/// Abstract base FB for components
{attribute 'enable_dynamic_creation' := ''}
{attribute 'reflection' := ''}
FUNCTION_BLOCK FB_ComponentBase IMPLEMENTS ITFComponent
VAR
	/// Unique ID of this instance (cam be used as index: P_ComponentPool.aComponents[iID]...)
	iId				: INT := -1;
	/// component active flag
	bActive			: BOOL;
	/// component state
	eState			: E_ComponentState;
	/// clear text info
	sClearText		: T_MaxString;
	/// last error debug info
	sLastError		: T_MaxString;	
	/// component type
	eTyp			: E_ComponentType;
	/// EventLog reference
	fbEventLog		: REFERENCE TO FB_EventLog;
	/// Last Event
	stLastEvent		: ST_Event;
	ptLastEvent		: POINTER TO ST_Event;
	
	
	/// Bereich
	eMachineArea	: E_MachineArea;
	/// component name
	sName			: STRING;
	/// BMK name
	sBMK			: STRING;
	/// path of this FB (e.g. for log: P_ComponentPool.fbVirtualMaster)
	{attribute 'no_init' := ''}
	{attribute 'instance-path' := ''}
	sPath			: STRING;	

END_VAR

///
/// Abstract base FB for components
/// TP/www.rmth.at/11.2014
///

/// Get's or set's a value indicating whether this component is active or not.
PROPERTY Active : BOOL
GET
Active := bActive;
END_GET
SET
bActive := Active;
sClearText := SEL(bActive, 'INACTIVE!', 'ACTIVE!');
END_SET
END_PROPERTY

PROPERTY BMK : STRING
GET
BMK := sBMK;
END_GET
SET
sBMK := BMK;
END_SET
END_PROPERTY

/// Get's value representing the component state.
PROPERTY ClearText : String
GET
ClearText := sClearText;
END_GET
END_PROPERTY

/// Unique component ID (cam be used as index: P_ComponentPool.aComponents[eID]...)
PROPERTY ID : INT
GET
ID := iId;
END_GET
SET
iID := Id;
END_SET
END_PROPERTY

/// Get's value representing the component state.
PROPERTY LastError : String
GET
LastError := sLastError;
END_GET
END_PROPERTY

PROPERTY MachineArea : E_MachineArea
GET
MachineArea := eMachineArea;
END_GET
SET
eMachineArea := MachineArea;
END_SET
END_PROPERTY

PROPERTY Name : STRING
GET
Name := sName;
END_GET
SET
sName := Name;
END_SET
END_PROPERTY

PROPERTY Path : String
GET
Path := sPath;
END_GET
END_PROPERTY

/// Reset component logic
{attribute 'object_name' := 'Reset'}
METHOD Reset
/// abstract base logic reset

sLastError := sEmpty;
MEMSET(ADR(stLastEvent), 0, SIZEOF(ST_EVENT));

// default: set state to ready
eState := E_ComponentState.eComponentState_ready;
END_METHOD

/// Run component logic
{attribute 'object_name' := 'Run'}
METHOD Run : E_ComponentState
/// abstract base logic run

// only rdy state may lead to run
IF eState = E_ComponentState.eComponentState_ready THEN
	eState := E_ComponentState.eComponentState_running;
END_IF

Run := eState;

IF stLastEvent.ePriority < E_Priority.ePriority_fault AND eState = E_ComponentState.eComponentState_error THEN
	WriteError(E_Event.eEvent_none, 'unbekannter Fehler');
END_IF
END_METHOD

/// Set EventLog reference
METHOD SetEventLogReference
VAR_IN_OUT
	/// HMI access provider.
	fbEventLogRef	: FB_EventLog;
END_VAR
fbEventLog REF= fbEventLogRef;
END_METHOD

/// Get's value representing the component state.
PROPERTY State : E_ComponentState
GET
State := eState;
END_GET
END_PROPERTY

/// Get's value representing the component state.
PROPERTY StateAsString : STRING
GET
CASE eState OF

	eComponentState_none :
		StateAsString := 'undefiniert';
	/// Component is resetting
	eComponentState_resetting:
		StateAsString := 'wird zurückgesetzt';
	/// Component is ready
	eComponentState_ready:
		StateAsString := 'ist bereit';
	/// Component is running
	eComponentState_running:
		StateAsString := 'wird ausgeführt';
	/// Component has error
	eComponentState_error:
		StateAsString := 'ist fehlerhaft';

END_CASE
END_GET
END_PROPERTY

PROPERTY Typ : E_ComponentType
GET
Typ := eTyp;
END_GET
END_PROPERTY

METHOD WriteError
VAR_INPUT
	Event			: E_Event;
	Description 	: T_MaxString;
END_VAR
WriteEvent(ePriority_fault, Event, Description, TRUE);
//eState := E_ComponentState.eComponentState_error;
END_METHOD

METHOD WriteEvent
VAR_INPUT
	Priority		: E_Priority;
	Event			: E_Event;
	Description 	: T_MaxString;
	Signalize			: BOOL;
END_VAR
VAR
	tmpItem: ST_Event;
END_VAR
// chk
IF NOT __ISVALIDREF(fbEventLog) THEN
	RETURN;
END_IF

tmpItem.eComponent := eTyp;
tmpItem.eEventID := Event;
tmpItem.eMachineArea := eMachineArea;
tmpItem.ePriority := Priority;
tmpItem.nComponentID := iId;
tmpItem.sDescription := Description;
tmpItem.bSignalize := Signalize;

IF 	ptLastEvent <> 0 AND_THEN
	ptLastEvent^.bIsRaised AND_THEN
   	tmpItem.eEventID = ptLastEvent^.eEventID AND_THEN
	tmpItem.sDescription = ptLastEvent^.sDescription AND_THEN 
	tmpItem.ePriority = ptLastEvent^.ePriority THEN 
	RETURN;
END_IF

ptLastEvent := fbEventLog.SetEvent(tmpItem);
stLastEvent := tmpItem;
END_METHOD

METHOD WriteInfo
VAR_INPUT
	Event			: E_Event;
	Description 	: T_MaxString;
END_VAR
WriteEvent(ePriority_info, Event, Description, FALSE);
END_METHOD

METHOD WriteWarning
VAR_INPUT
	Event			: E_Event;
	Description 	: T_MaxString;
	Signal			: BOOL;
END_VAR
VAR
	tmpItem			: ST_Event;
END_VAR
WriteEvent(ePriority_warning, Event, Description, Signal);
END_METHOD

END_FUNCTION_BLOCK

(* stored: Version 1.1.0.1, ProductVersion 3.1.4022.10
   POU FB_ComponentBase: Id {c18f24bd-a664-4b00-87c6-35388a9e2c13}, SpecialFunc None
   Folder Properties: Id {2d8306c8-917b-4b20-9aa7-5415be6cad83}
   Folder Utilities: Id {18cd2ad0-5a5a-4e5f-92e4-b0238b542ab5}
   Property Active: Id {ad08f73b-d076-4ffc-a47f-109b9002f3f0}
   Get Get: Id {8dd8e62e-65cf-4eae-a985-79199664088e}
   Set Set: Id {1d543709-b1d6-4f2d-af6c-97246f4599c2}
   Property BMK: Id {3e8ee465-5189-4f2f-9d15-0d6a660f5497}
   Get Get: Id {01c92174-19fd-4b80-81d2-175c5750d2bc}
   Set Set: Id {b8ef3cfc-b534-4fcd-97bc-b47816b7b27a}
   Property ClearText: Id {56ead6a6-eff4-4858-8e9e-da8349489d0c}
   Get Get: Id {1fa5bb79-05f3-4363-a22b-26790775d81b}
   Property ID: Id {7adf225e-7442-4f77-874e-8de91565912f}
   Get Get: Id {ddac6993-c733-47b1-a445-f075002f8c38}
   Set Set: Id {9987bba1-8297-46ec-8910-10e8ca7a5cd6}
   Property LastError: Id {06cb7fc4-a4a0-4ce5-a61e-ff39359d5455}
   Get Get: Id {fbc8f7e9-e26a-44c8-a99b-ddf89c43d61b}
   Property MachineArea: Id {5002829a-7be9-4fd2-bdb1-4f471524ec33}
   Get Get: Id {b1107982-d402-48e8-82e1-34f3ffa3cd58}
   Set Set: Id {3ad4b5e6-3b5e-468e-b88a-52a5ed7a2777}
   Property Name: Id {97507556-cbd6-4656-a4b4-7ef03ea2ff1e}
   Get Get: Id {5bc1be01-8584-43a7-b2c4-089d7b7d1290}
   Set Set: Id {cdf272ad-e29a-4767-ad58-2d41f72fa33a}
   Property Path: Id {f15c3da9-69b6-42be-b750-91438e4fc191}
   Get Get: Id {c3c5d9a1-7c3c-440f-abee-27056ac72a80}
   Method Reset: Id {7800391a-478c-4265-bd45-1c25f898c8f4}
   Method Run: Id {04530f9f-040a-4517-8bda-6e0d48f73e41}
   Method SetEventLogReference: Id {452527ba-597e-4211-8fa1-0bbb9e3c7ffb}
   Property State: Id {d68fb6ae-0af8-44c3-bb4d-32b1388481b9}
   Get Get: Id {b4088dcc-e43a-4064-b0df-93c47386d3d2}
   Property StateAsString: Id {bffb55f1-1ef3-4369-ab66-e92ce785efbd}
   Get Get: Id {3dd43a60-ec91-4906-860b-12629fae2ae4}
   Property Typ: Id {987dd2cf-7ace-4cc4-856e-8b41f907e2c3}
   Get Get: Id {9fd10945-acfb-45ad-818f-6e98f300ba25}
   Method WriteError: Id {a92622fe-49fc-4553-8379-a99997764084}
   Method WriteEvent: Id {583be540-6251-46c4-8656-e5b754778d2f}
   Method WriteInfo: Id {c2be943a-77e2-432b-be2b-8003842ed1ca}
   Method WriteWarning: Id {05cae7cb-6c8d-4876-827e-346c099d6a8b} *)
